TYPE ST_DB_OACDataCtrl :
STRUCT
	bCreateDataReq				: BOOL;	(* C *)
	bReadDataReq				: BOOL;	(* R *)
	bUpdateDataReq				: BOOL;	(* U *)
	bDeleteDataReq				: BOOL;	(* D *)

	sFileCodeName				: T_MaxString;
	
	bBlockRecord				: BOOL;
	bRestored					: BOOL;

	stOACStatusDB				: ST_OUTER_Status;

	bDone						: BOOL;
	bError						: BOOL;
	nErrorID					: UDINT;

END_STRUCT
END_TYPE

(* stored: Version 1.1.0.1
   DUT ST_DB_OACDataCtrl: Id {bd0eb1ae-7677-4e37-a200-7ff3ad801833} *)
